{attribute 'GeneratedUsingTerminal: ER2339-0021-0018'}
{attribute addProperty BoxType "ER2339-0021-0018"}
{attribute addProperty Id "AoeNetIdAT %I*.TcoAmsNetId0StateAT %I*UINT2"}
{attribute addProperty CRC "131947802"}
{attribute addProperty Size "2"}
TYPE InfoData_07DD5D1A :
STRUCT
	{attribute addProperty Name "AoeNetId"}
	AoeNetId AT %I* : .TcoAmsNetId;
	{attribute addProperty Name "State"}
	State AT %I* : UINT;
END_STRUCT
END_TYPE

(* stored: Version 1.2.0.0, ProductVersion 3.1.4024.9
   DUT InfoData_07DD5D1A: Id {c3abcdc8-de36-4b27-b172-0ad136fb51d5} *)
